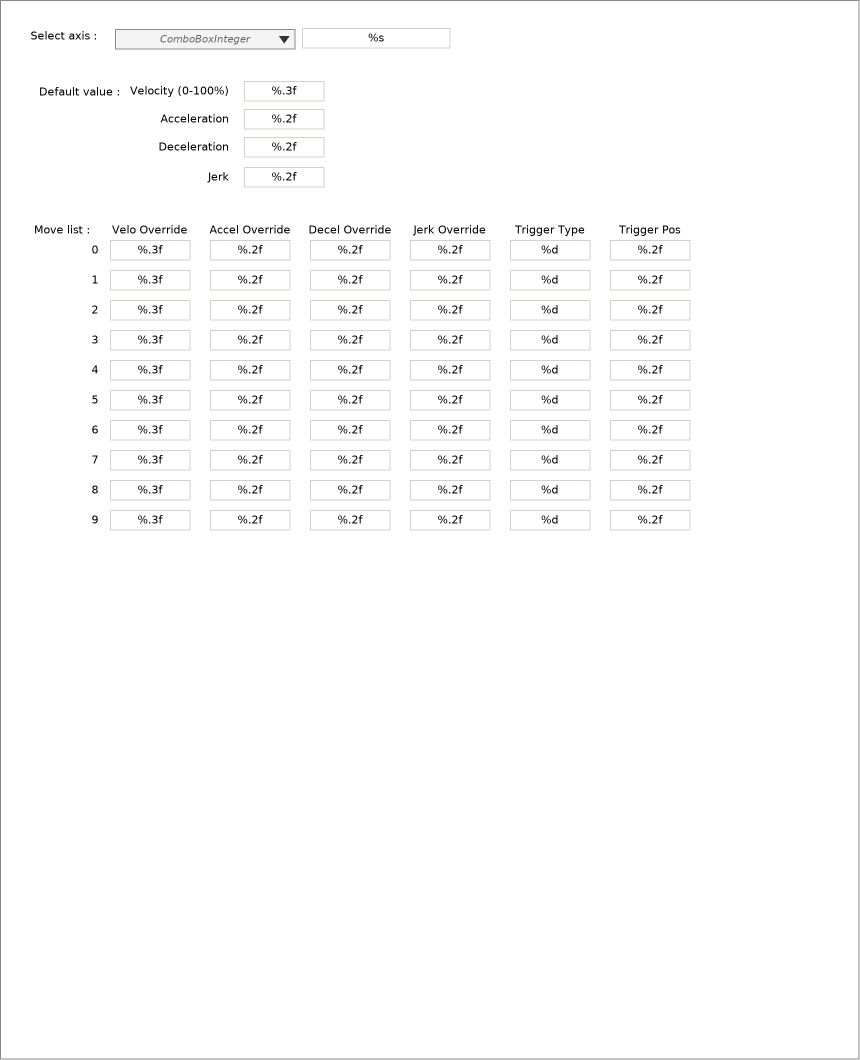
VISUALIZATION VISU_LinearConfigArray  // 860x1060
    Label (15,220 94x20), "Move list :"
    Label (12,82 135x20), "Default value :"
    Label (22,21 84x30), "Select axis :"
    Label (132,81 100x20), "Velocity (0-100%)"
    Label (132,109 100x20), "Acceleration"
    Label (132,137 100x20), "Deceleration"
    Label (132,167 100x20), "Jerk"
    Textfield (244,81 80x20), "%.3f", text variable: PERS.recipeList.linearAxis[HMI.iSelectAxis].defProfile.lrVelocity
        OnMouseDown: write the text variable via Default
    Textfield (244,109 80x20), "%.2f", text variable: PERS.recipeList.linearAxis[HMI.iSelectAxis].defProfile.lrAccel
        OnMouseDown: write the text variable via Default
    Textfield (244,137 80x20), "%.2f", text variable: PERS.recipeList.linearAxis[HMI.iSelectAxis].defProfile.lrDecel
        OnMouseDown: write the text variable via Default
    Textfield (244,167 80x20), "%.2f", text variable: PERS.recipeList.linearAxis[HMI.iSelectAxis].defProfile.lrJerk
        OnMouseDown: write the text variable via Default
    Label (100,220 100x20), "Velo Override"
    Label (200,220 100x20), "Accel Override"
    Label (300,220 100x20), "Decel Override"
    Label (400,220 100x20), "Jerk Override"
    Label (500,220 100x20), "Trigger Type"
    Label (600,220 100x20), "Trigger Pos"
    Textfield (110,240 80x20), "%.3f", text variable: PERS.recipeList.linearAxis[HMI.iSelectAxis].movesList[0].lrVelocity
        OnMouseDown: write the text variable via Default
    Label (80,240 30x20), "0"
    Textfield (210,240 80x20), "%.2f", text variable: PERS.recipeList.linearAxis[HMI.iSelectAxis].movesList[0].lrAccel
        OnMouseDown: write the text variable via Default
    Textfield (310,240 80x20), "%.2f", text variable: PERS.recipeList.linearAxis[HMI.iSelectAxis].movesList[0].lrDecel
        OnMouseDown: write the text variable via Default
    Textfield (410,240 80x20), "%.2f", text variable: PERS.recipeList.linearAxis[HMI.iSelectAxis].movesList[0].lrJerk
        OnMouseDown: write the text variable via Default
    Textfield (510,240 80x20), "%d", text variable: PERS.recipeList.linearAxis[HMI.iSelectAxis].movesList[0].TriggerType
        OnMouseDown: write the text variable via Default
    Textfield (610,240 80x20), "%.2f", text variable: PERS.recipeList.linearAxis[HMI.iSelectAxis].movesList[0].TriggerPos
        OnMouseDown: write the text variable via Default
    Textfield (110,270 80x20), "%.3f", text variable: PERS.recipeList.linearAxis[HMI.iSelectAxis].movesList[1].lrVelocity
        OnMouseDown: write the text variable via Default
    Label (80,270 30x20), "1"
    Textfield (210,270 80x20), "%.2f", text variable: PERS.recipeList.linearAxis[HMI.iSelectAxis].movesList[1].lrAccel
        OnMouseDown: write the text variable via Default
    Textfield (310,270 80x20), "%.2f", text variable: PERS.recipeList.linearAxis[HMI.iSelectAxis].movesList[1].lrDecel
        OnMouseDown: write the text variable via Default
    Textfield (410,270 80x20), "%.2f", text variable: PERS.recipeList.linearAxis[HMI.iSelectAxis].movesList[1].lrJerk
        OnMouseDown: write the text variable via Default
    Textfield (510,270 80x20), "%d", text variable: PERS.recipeList.linearAxis[HMI.iSelectAxis].movesList[1].TriggerType
        OnMouseDown: write the text variable via Default
    Textfield (610,270 80x20), "%.2f", text variable: PERS.recipeList.linearAxis[HMI.iSelectAxis].movesList[1].TriggerPos
        OnMouseDown: write the text variable via Default
    Textfield (110,300 80x20), "%.3f", text variable: PERS.recipeList.linearAxis[HMI.iSelectAxis].movesList[2].lrVelocity
        OnMouseDown: write the text variable via Default
    Label (80,300 30x20), "2"
    Textfield (210,300 80x20), "%.2f", text variable: PERS.recipeList.linearAxis[HMI.iSelectAxis].movesList[2].lrAccel
        OnMouseDown: write the text variable via Default
    Textfield (310,300 80x20), "%.2f", text variable: PERS.recipeList.linearAxis[HMI.iSelectAxis].movesList[2].lrDecel
        OnMouseDown: write the text variable via Default
    Textfield (410,300 80x20), "%.2f", text variable: PERS.recipeList.linearAxis[HMI.iSelectAxis].movesList[2].lrJerk
        OnMouseDown: write the text variable via Default
    Textfield (510,300 80x20), "%d", text variable: PERS.recipeList.linearAxis[HMI.iSelectAxis].movesList[2].TriggerType
        OnMouseDown: write the text variable via Default
    Textfield (610,300 80x20), "%.2f", text variable: PERS.recipeList.linearAxis[HMI.iSelectAxis].movesList[2].TriggerPos
        OnMouseDown: write the text variable via Default
    Textfield (110,330 80x20), "%.3f", text variable: PERS.recipeList.linearAxis[HMI.iSelectAxis].movesList[3].lrVelocity
        OnMouseDown: write the text variable via Default
    Label (80,330 30x20), "3"
    Textfield (210,330 80x20), "%.2f", text variable: PERS.recipeList.linearAxis[HMI.iSelectAxis].movesList[3].lrAccel
        OnMouseDown: write the text variable via Default
    Textfield (310,330 80x20), "%.2f", text variable: PERS.recipeList.linearAxis[HMI.iSelectAxis].movesList[3].lrDecel
        OnMouseDown: write the text variable via Default
    Textfield (410,330 80x20), "%.2f", text variable: PERS.recipeList.linearAxis[HMI.iSelectAxis].movesList[3].lrJerk
        OnMouseDown: write the text variable via Default
    Textfield (510,330 80x20), "%d", text variable: PERS.recipeList.linearAxis[HMI.iSelectAxis].movesList[3].TriggerType
        OnMouseDown: write the text variable via Default
    Textfield (610,330 80x20), "%.2f", text variable: PERS.recipeList.linearAxis[HMI.iSelectAxis].movesList[3].TriggerPos
        OnMouseDown: write the text variable via Default
    Textfield (110,360 80x20), "%.3f", text variable: PERS.recipeList.linearAxis[HMI.iSelectAxis].movesList[4].lrVelocity
        OnMouseDown: write the text variable via Default
    Label (80,360 30x20), "4"
    Textfield (210,360 80x20), "%.2f", text variable: PERS.recipeList.linearAxis[HMI.iSelectAxis].movesList[4].lrAccel
        OnMouseDown: write the text variable via Default
    Textfield (310,360 80x20), "%.2f", text variable: PERS.recipeList.linearAxis[HMI.iSelectAxis].movesList[4].lrDecel
        OnMouseDown: write the text variable via Default
    Textfield (410,360 80x20), "%.2f", text variable: PERS.recipeList.linearAxis[HMI.iSelectAxis].movesList[4].lrJerk
        OnMouseDown: write the text variable via Default
    Textfield (510,360 80x20), "%d", text variable: PERS.recipeList.linearAxis[HMI.iSelectAxis].movesList[4].TriggerType
        OnMouseDown: write the text variable via Default
    Textfield (610,360 80x20), "%.2f", text variable: PERS.recipeList.linearAxis[HMI.iSelectAxis].movesList[4].TriggerPos
        OnMouseDown: write the text variable via Default
    Textfield (110,390 80x20), "%.3f", text variable: PERS.recipeList.linearAxis[HMI.iSelectAxis].movesList[5].lrVelocity
        OnMouseDown: write the text variable via Default
    Label (80,390 30x20), "5"
    Textfield (210,390 80x20), "%.2f", text variable: PERS.recipeList.linearAxis[HMI.iSelectAxis].movesList[5].lrAccel
        OnMouseDown: write the text variable via Default
    Textfield (310,390 80x20), "%.2f", text variable: PERS.recipeList.linearAxis[HMI.iSelectAxis].movesList[5].lrDecel
        OnMouseDown: write the text variable via Default
    Textfield (410,390 80x20), "%.2f", text variable: PERS.recipeList.linearAxis[HMI.iSelectAxis].movesList[5].lrJerk
        OnMouseDown: write the text variable via Default
    Textfield (510,390 80x20), "%d", text variable: PERS.recipeList.linearAxis[HMI.iSelectAxis].movesList[5].TriggerType
        OnMouseDown: write the text variable via Default
    Textfield (610,390 80x20), "%.2f", text variable: PERS.recipeList.linearAxis[HMI.iSelectAxis].movesList[5].TriggerPos
        OnMouseDown: write the text variable via Default
    Textfield (110,420 80x20), "%.3f", text variable: PERS.recipeList.linearAxis[HMI.iSelectAxis].movesList[6].lrVelocity
        OnMouseDown: write the text variable via Default
    Label (80,420 30x20), "6"
    Textfield (210,420 80x20), "%.2f", text variable: PERS.recipeList.linearAxis[HMI.iSelectAxis].movesList[6].lrAccel
        OnMouseDown: write the text variable via Default
    Textfield (310,420 80x20), "%.2f", text variable: PERS.recipeList.linearAxis[HMI.iSelectAxis].movesList[6].lrDecel
        OnMouseDown: write the text variable via Default
    Textfield (410,420 80x20), "%.2f", text variable: PERS.recipeList.linearAxis[HMI.iSelectAxis].movesList[6].lrJerk
        OnMouseDown: write the text variable via Default
    Textfield (510,420 80x20), "%d", text variable: PERS.recipeList.linearAxis[HMI.iSelectAxis].movesList[6].TriggerType
        OnMouseDown: write the text variable via Default
    Textfield (610,420 80x20), "%.2f", text variable: PERS.recipeList.linearAxis[HMI.iSelectAxis].movesList[6].TriggerPos
        OnMouseDown: write the text variable via Default
    Textfield (110,450 80x20), "%.3f", text variable: PERS.recipeList.linearAxis[HMI.iSelectAxis].movesList[7].lrVelocity
        OnMouseDown: write the text variable via Default
    Label (80,450 30x20), "7"
    Textfield (210,450 80x20), "%.2f", text variable: PERS.recipeList.linearAxis[HMI.iSelectAxis].movesList[7].lrAccel
        OnMouseDown: write the text variable via Default
    Textfield (310,450 80x20), "%.2f", text variable: PERS.recipeList.linearAxis[HMI.iSelectAxis].movesList[7].lrDecel
        OnMouseDown: write the text variable via Default
    Textfield (410,450 80x20), "%.2f", text variable: PERS.recipeList.linearAxis[HMI.iSelectAxis].movesList[7].lrJerk
        OnMouseDown: write the text variable via Default
    Textfield (510,450 80x20), "%d", text variable: PERS.recipeList.linearAxis[HMI.iSelectAxis].movesList[7].TriggerType
        OnMouseDown: write the text variable via Default
    Textfield (610,450 80x20), "%.2f", text variable: PERS.recipeList.linearAxis[HMI.iSelectAxis].movesList[7].TriggerPos
        OnMouseDown: write the text variable via Default
    Textfield (110,480 80x20), "%.3f", text variable: PERS.recipeList.linearAxis[HMI.iSelectAxis].movesList[8].lrVelocity
        OnMouseDown: write the text variable via Default
    Label (80,480 30x20), "8"
    Textfield (210,480 80x20), "%.2f", text variable: PERS.recipeList.linearAxis[HMI.iSelectAxis].movesList[8].lrAccel
        OnMouseDown: write the text variable via Default
    Textfield (310,480 80x20), "%.2f", text variable: PERS.recipeList.linearAxis[HMI.iSelectAxis].movesList[8].lrDecel
        OnMouseDown: write the text variable via Default
    Textfield (410,480 80x20), "%.2f", text variable: PERS.recipeList.linearAxis[HMI.iSelectAxis].movesList[8].lrJerk
        OnMouseDown: write the text variable via Default
    Textfield (510,480 80x20), "%d", text variable: PERS.recipeList.linearAxis[HMI.iSelectAxis].movesList[8].TriggerType
        OnMouseDown: write the text variable via Default
    Textfield (610,480 80x20), "%.2f", text variable: PERS.recipeList.linearAxis[HMI.iSelectAxis].movesList[8].TriggerPos
        OnMouseDown: write the text variable via Default
    Textfield (110,510 80x20), "%.3f", text variable: PERS.recipeList.linearAxis[HMI.iSelectAxis].movesList[9].lrVelocity
        OnMouseDown: write the text variable via Default
    Label (80,510 30x20), "9"
    Textfield (210,510 80x20), "%.2f", text variable: PERS.recipeList.linearAxis[HMI.iSelectAxis].movesList[9]
        OnMouseDown: write the text variable via Default
    Textfield (310,510 80x20), "%.2f", text variable: PERS.recipeList.linearAxis[HMI.iSelectAxis].movesList[9].lrDecel
        OnMouseDown: write the text variable via Default
    Textfield (410,510 80x20), "%.2f", text variable: PERS.recipeList.linearAxis[HMI.iSelectAxis].movesList[9].lrJerk
        OnMouseDown: write the text variable via Default
    Textfield (510,510 80x20), "%d", text variable: PERS.recipeList.linearAxis[HMI.iSelectAxis].movesList[9].TriggerType
        OnMouseDown: write the text variable via Default
    Textfield (610,510 80x20), "%.2f", text variable: PERS.recipeList.linearAxis[HMI.iSelectAxis].movesList[9].TriggerPos
        OnMouseDown: write the text variable via Default
    ComboBoxInteger (115,29 180x20), variable: HMI.iSelectAxis
    Textfield (302,28 148x20), "%s", text variable: TO_STRING(HMI.iSelectAxis)
END_VISUALIZATION

(* stored: Version 1.1.0.1, ProductVersion 3.1.4024.6
   Visu VISU_LinearConfigArray: Id {53576da3-4487-46ff-a2bf-be3d853ced4e} *)
